(* CoDeSys 2.3 export: MBSTEPE.EXP *)

(* Data type *)
TYPE MBStepE :
(
    StepSelect,
    MV110Read,
    MU110Write
);
END_TYPE
